{attribute 'qualified_only'}
VAR_GLOBAL
	Action1:BOOL;
	Action2:BOOL;
	Action3:BOOL;
	Action4:BOOL;
END_VAR

(* stored: Version 1.1.0.1
   GVL HMI: Id {b996835f-f8a5-4024-a4ba-b87619fe1b4e} *)
